FUNCTION_BLOCK FB_FlowScaling
VAR_INPUT
	nRawInput : INT;
	stFlowParams : ST_FlowScale; 
END_VAR
VAR_OUTPUT
	fScaledFlow : LREAL; 
END_VAR
VAR
	fRawInput 				: LREAL;
	fTempInput 				: LREAL;
	fTempOutput 			: LREAL;
END_VAR

fRawInput := INT_TO_LREAL(nRawInput);

fTempInput := fRawInput - stFlowParams.fNeutralFlowInput;

IF fTempInput > stFlowParams.fNeutralDeadband THEN
	fTempOutput := fTempInput/(stFlowParams.fMaxFlowInput - stFlowParams.fNeutralFlowInput);
ELSIF fTempInput < -stFlowParams.fNeutralDeadband THEN	
	fTempOutput := fTempInput/(stFlowParams.fNeutralFlowInput - stFlowParams.fMinFlowInput);
ELSE
	fTempOutput := 0.0;
END_IF

fScaledFlow := LIMIT(stFlowParams.fMinFlowOutput, fTempOutput*150.0, stFlowParams.fMaxFlowOutput);

END_FUNCTION_BLOCK

(* stored: Version 1.1.0.1, ProductVersion 3.1.4024.12
   POU FB_FlowScaling: Id {5b0a1ced-bfac-4021-b133-029f32b502b6}, SpecialFunc None *)
